FUNCTION alg_a_Dresetled : BOOL
VAR_INPUT
	state: STATE;
END_VAR

alg_a_Dresetled := FALSE;

END_FUNCTION

(* stored: Version 1.1.0.1, ProductVersion 3.1.4022.18
   POU alg_a_Dresetled: Id {81df0fa5-4f48-486d-9589-c9cf5214a40b}, SpecialFunc None *)
